// TIA Portal V20 export
TYPE "typeSequenceControlNode"
// stored: Namespace Unit1.Em1
   STRUCT
      jobs : "LAF_typeJobs";
      sequence : "LAF_typeSequence";
      selectJobStatus { S7_SetPoint := 'True'} : Array[0..10] of "LAF_typeJobStatus";
      "step" : "LER_typeStep";
      jobInterface : "Unit1.Em1.typeSequenceControlNodeJobInterface";
      homeCheck : "Unit1.Em1.typeSequenceControlNodeHomeCheck";
   END_STRUCT;
   // // "step".action1[101] : Step[101] : JOB[1] Condition
   // // "step".action1[110] : Step[110] : Clamp Z Up
   // // "step".action1[120] : Step[120] : Clamp Unit Mover Backward
   // // "step".action1[130] : Step[130] : Clamp Left, Right Open
   // // "step".action1[140] : Step[140] : Clamp Mover Open
   // // "step".action1[180] : Step[180] : Lift Down
   // // "step".action1[190] : Step[190] : JOB[1] Step End
   // // "step".action1[201] : Step[201] : JOB[2] Condition
   // // "step".action1[210] : Step[210] : Clamp Unit Mover Forward
   // // "step".action1[220] : Step[220] : Clamp Mover Close
   // // "step".action1[230] : Step[230] : Clamp Left, Right Close
   // // "step".action1[231] : Step[231] : Stacker #2 NG Box [Unclamp Request] => Stack #2
   // // "step".action1[240] : Step[240] : Clamp Unit Mover Backward
   // // "step".action1[290] : Step[290] : JOB[2] Step End
   // // "step".action1[301] : Step[301] : JOB[3] Condition
   // // "step".action1[310] : Step[310] : Clamp Unit Mover Forward
   // // "step".action1[320] : Step[320] : Clamp Z Down
   // // "step".action1[330] : Step[330] : Clamp Left, Right Open
   // // "step".action1[340] : Step[340] : Clamp Mover Open
   // // "step".action1[350] : Step[350] : Clamp Z Up
   // // "step".action1[360] : Step[360] : Clamp Unit Mover Backward
   // // "step".action1[390] : Step[390] : JOB[3] Step End
   // // "step".transition1[101] : Step[101] : JOB[1] Condition
   // // "step".transition1[110] : Step[110] : Clamp Z Up
   // // "step".transition1[120] : Step[120] : Clamp Unit Mover Backward
   // // "step".transition1[130] : Step[130] : Clamp Left, Right Open
   // // "step".transition1[140] : Step[140] : Clamp Mover Open
   // // "step".transition1[180] : Step[180] : Lift Down
   // // "step".transition1[190] : Step[190] : JOB[1] Step End
   // // "step".transition1[201] : Step[201] : JOB[2] Condition
   // // "step".transition1[210] : Step[210] : Clamp Unit Mover Forward
   // // "step".transition1[220] : Step[220] : Clamp Mover Close
   // // "step".transition1[230] : Step[230] : Clamp Left, Right Close
   // // "step".transition1[231] : Step[231] : Stacker #2 NG Box [Unclamp Request] => Stack #2
   // // "step".transition1[240] : Step[240] : Clamp Unit Mover Backward
   // // "step".transition1[290] : Step[290] : JOB[2] Step End
   // // "step".transition1[301] : Step[301] : JOB[3] Condition
   // // "step".transition1[310] : Step[310] : Clamp Unit Mover Forward
   // // "step".transition1[320] : Step[320] : Clamp Z Down
   // // "step".transition1[330] : Step[330] : Clamp Left, Right Open
   // // "step".transition1[340] : Step[340] : Clamp Mover Open
   // // "step".transition1[350] : Step[350] : Clamp Z Up
   // // "step".transition1[360] : Step[360] : Clamp Unit Mover Backward
   // // "step".transition1[390] : Step[390] : JOB[3] Step End
END_TYPE
